Staubli VAL3: get_num.pgx

public program get_num(string& x_sItem[] (dimensions=1), num x_nIndex (dimensions=1))
  local string l_sKey
  local num i
begin
  // OUTPUT
  // start from the first
  l_sKey=first(cCount)
  // search it
  while l_sKey!=""
    x_sItem=l_sKey
    l_sKey=next(cCount[l_sKey])
    if i==x_nIndex
      return
    else
      i=i+1
    endIf
  endWhile
  // start from the first
  l_sKey=first(aCount)
  while l_sKey!=""
    x_sItem=l_sKey
    l_sKey=next(aCount[l_sKey])
    if i==x_nIndex
      return
    else
      i=i+1
    endIf
  endWhile
end
